(* PLC project SWPR1010_A1_0_FBD.project, CODESYS CODESYS V3.5 SP16 Patch 6 *)
(* stored: creationDateTime 2025-08-14T16:12:58.6358024, modificationDateTime 1601-01-01T02:00:00 *)

(* Created by : Serdar Temeltasi, Date created : 06.03.2025 Description : Checks whether charge button is pressed *)
FUNCTION_BLOCK _FB_MC_Chk_Chrg_Btn
  VAR_INPUT
    S_Bwd_Lft_Chrg_Btn : BOOL;
    S_Stop_Lft_Chrg : BOOL;
  END_VAR
  VAR_OUTPUT
    S_Chrg_Btn : BOOL;
  END_VAR
  VAR
    S_AC_Chrg_On_Btn : BOOL;
    R_TRIG_0 : R_TRIG;
    TON_0 : TON;
    RS_0 : RS;
    TON_1 : TON;
    R_TRIG_1 : R_TRIG;
  END_VAR
  VAR  (* added by the conversion: wires and edge detectors of the diagram *)
    _OR13_OUT : BOOL;
  END_VAR

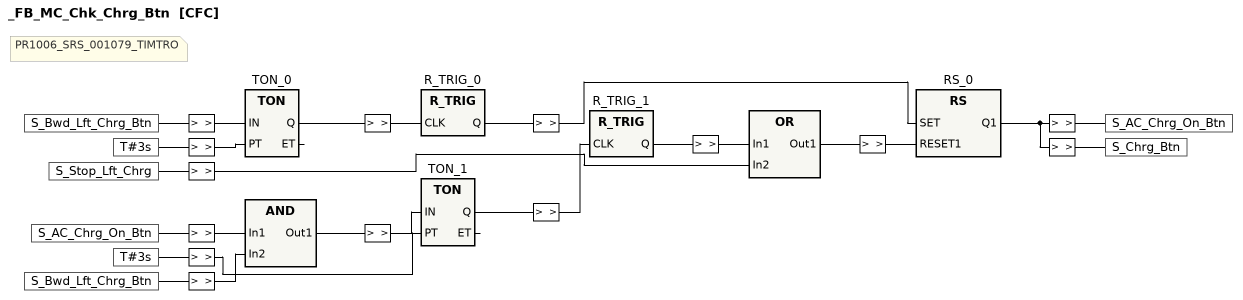
(* CFC diagram, written out as Structured Text *)
(* PR1006_SRS_001079_TIMTRO *)
TON_0(IN := S_Bwd_Lft_Chrg_Btn, PT := T#3s);
R_TRIG_0(CLK := TON_0.Q);
S_AC_Chrg_On_Btn := RS_0.Q1;
S_Chrg_Btn := RS_0.Q1;
_OR13_OUT := R_TRIG_1.Q OR S_Stop_Lft_Chrg;
RS_0(SET := R_TRIG_0.Q, RESET1 := _OR13_OUT);
R_TRIG_1(CLK := TON_1.Q);
TON_1(IN := S_AC_Chrg_On_Btn AND S_Bwd_Lft_Chrg_Btn, PT := T#3s);
END_FUNCTION_BLOCK
